(* CODESYS project jt808.20211124.1.project

Project tree, tasks and I/O mapping:
  MIC7001 : Changsha-Cyber-MI-linux, Changsha Cyber-MI Co., Ltd., version 3.5.10.40
    application Application
      libraries: Standard, * (System); CAA Types Extern, * (CAA Technical Workgroup); CAA Callback Extern, * (CAA Technical Workgroup); SysMem, * (System); SysTypes Interfaces, * (System); SysTime, * (System); CAA DTUtil Extern, 3.5.12.0 (CAA Technical Workgroup); CAA Real Time Clock Extern, 3.5.10.0 (CAA Technical Workgroup); CAN API, 1.0.0.3 (3S - Smart Software Solutions GmbH); SysFile, 3.5.15.0 (System); AC_DataLog, 3.5.14.0 (3S - Smart Software Solutions GmbH); CAA Net Base Services, 3.5.15.0 (CAA Technical Workgroup); CAA Memory, 3.5.12.0 (CAA Technical Workgroup); CAA SerialCom, 3.5.15.0 (CAA Technical Workgroup); MIC7001 base library, 1.0 (Cyber-MI.com); Util, 3.5.15.0 (System); CAA Can Low Level Imp Extern, 3.5.11.0 (CAA Technical Workgroup); CAA Can Low Level Extern, 3.5.15.0 (CAA Technical Workgroup); VisuDialogs, * (System); CmpBitmapPool, * (System); CAA File, 3.5.15.0 (CAA Technical Workgroup); IODrvEtherCAT, 3.5.15.50 (3S - Smart Software Solutions GmbH); SysShm, 3.5.8.0 (System)
      task VISU_TASK (cyclic, interval 100 ms, priority 31) calls prg_gps, prg_jt808, VisuElems.Visu_Prg
      trace Trace (task task_10ms): GVL_IO.remote_di, GVL_IO.b_mode_remote
      06_jt808/
        programs/
          program prg_jt808 [ST]: send_to_server, read_from_server, init
          program prg_gps [ST]
        Structs/
          data type stShmJT808Down
          data type stLocationExt
          data type stShmJT808Up
          data type stLocationBase
          data type stCanFrm
          data type nmeaTIME
          data type nmeaGPRMC
        functions/
          function get_sub_string_1 [ST]
          function nmea_parse_time [ST]
          function nmea_parse_date [ST]
          function get_latlon_from_str [ST]
          function nmea_parse_GPRMC [ST]
        functionblocks/
          function block Com_gps [ST]
    SoftMotion General Axis Pool
  libraries: CmpBitmapPool, * (System)
  image pool ImagePool_1
  image pool ImagePool
  5ce3da45-db07-42e7-a21c-a00fff4ed8f6|C:\Users\RJST\Desktop\bmp1.png
  text list GlobalTextList
*)

// MIC7001/Application/06_jt808/Structs/stShmJT808Down
TYPE stShmJT808Down :  // JT808下行数据
STRUCT
	location_interval:DINT;  // 位置信息发送间隔， 单位： ms
	ctrl : DINT;   // 车辆控制命令
END_STRUCT
END_TYPE

// MIC7001/Application/06_jt808/Structs/stLocationExt
TYPE stLocationExt :
STRUCT
	km_all: DINT;  // km all
	fuel:INT;   // fuel meter
	speed: INT;  // speed can
	lac:DINT; 
	cid:DINT;
	fuel_trip:DINT; // 本行程油耗
	fuel_all:DINT; 
	fuel_r_h:DINT;  // 0.05L/h
	fuel_r_l:DINT;  //  1/512Km/L
END_STRUCT
END_TYPE

// MIC7001/Application/06_jt808/Structs/stShmJT808Up
TYPE stShmJT808Up :   // 发送到服务器的上行数据
STRUCT
    location:stLocationBase;
	loc_ext:stLocationExt;
	can_data:stCanFrm;
END_STRUCT
END_TYPE

// MIC7001/Application/06_jt808/Structs/stLocationBase
TYPE stLocationBase :
STRUCT
	warning : UDINT;
    status : UDINT;
    latitude : DINT;
    longitude : DINT;
    altitude : INT;
    speed : INT;
    bearing : INT;
    asc_time :ARRAY[0..5] OF BYTE;  // ascii YYMMDDhhmmss (GMT+8)
END_STRUCT
END_TYPE

// MIC7001/Application/06_jt808/Structs/stCanFrm
TYPE stCanFrm :
STRUCT
	sn:UDINT;  // 每次更新内容后加一，用于通知底层发送程序
	id:UDINT;  //  CAN id
	data:ARRAY[0..7] OF BYTE;  // 8个字节 数据
END_STRUCT
END_TYPE

// MIC7001/Application/06_jt808/Structs/nmeaTIME
TYPE nmeaTIME :
STRUCT
	year:DINT;
	month:DINT;
	day:DINT;
	hour:DINT;
	minute:DINT;
	second:DINT;
	hsecond:DINT;
END_STRUCT
END_TYPE

// MIC7001/Application/06_jt808/Structs/nmeaGPRMC
TYPE nmeaGPRMC :
STRUCT
	utc : nmeaTIME;
	status : STRING(1);
	lat : REAL;
	ns : STRING(1);
	lon : REAL;
	ew : STRING(1);
	speed : REAL;
	direction : REAL;
	declination : REAL;
	declin_ew : STRING(1);
	mode : STRING(1);
END_STRUCT
END_TYPE

// MIC7001/Application/06_jt808/programs/prg_gps
PROGRAM prg_gps
VAR  
	filename:STRING(256) := '/tmp/connect_server.txt';
	hFile: RTS_IEC_HANDLE := 0;
	udiOpenError: RTS_IEC_RESULT;
	connect_open_flag :BOOL := TRUE;
	
	gps :Com_gps;
	com_handle :CAA.HANDLE; 
	packGPRMC : nmeaGPRMC;
	buf:STRING(255);
	gps_ok:BOOL := FALSE;
END_VAR

// 判断后端PPP网络是否连通，如果已经连通，则会同步网络时间
IF connect_open_flag THEN
	hFile := sysfileopen(szFile := filename, am := sysfile.AM_READ, pResult:= ADR(udiOpenError));
	IF hFile = RTS_INVALID_HANDLE THEN
		RETURN;
	END_IF
	
	hFile := MIC7001_BASE.close_file(hFile := hFile);
	connect_open_flag := FALSE;
END_IF

gps(xEnable := TRUE, com_hand := com_handle, gps_str => buf); 

nmea_parse_GPRMC(buf, SIZEOF(buf), ADR(packGPRMC));

IF packGPRMC.status = 'A' THEN
	gps_ok := TRUE;
ELSE
	gps_ok := FALSE;
END_IF

END_PROGRAM

// MIC7001/Application/06_jt808/functions/nmea_parse_GPRMC
FUNCTION nmea_parse_GPRMC : bool
VAR_INPUT
    buff : STRING(255);
	buff_sz : DINT;
	pack : POINTER TO nmeaGPRMC;
END_VAR
VAR
	str:STRING(255);
	rc :BOOL;
	checksum : DINT;	
END_VAR

nmea_parse_GPRMC := FALSE;

str := get_sub_string(buff, '$$', ',', 1);   //check 'GPRMC'
IF str <> 'GPRMC' THEN
	RETURN;
END_IF

//find time
str := get_sub_string(buff, ',', ',', 1);  
IF len(str) < len('hhmmss')  THEN
	RETURN;  //format error	
END_IF
IF NOT nmea_parse_time(str, ADR(pack^.utc)) THEN
	RETURN;
END_IF

//find status
str := get_sub_string(buff, ',', ',', 2);  
IF len(str)<1 THEN
	RETURN; //format error
END_IF
pack^.status := str;

//find lat
str := get_sub_string(buff, ',', ',', 3);  
IF len(str)<1 THEN
	RETURN; //format error
END_IF
pack^.lat := get_latlon_from_str(str);

//find ns
str := get_sub_string(buff, ',', ',', 4); 
IF len(str)<1 THEN
	RETURN; //format error
END_IF
pack^.ns := str;

//find lon
str := get_sub_string(buff, ',', ',', 5); 
IF len(str)<1 THEN
	RETURN; //format error
END_IF
pack^.lon := get_latlon_from_str(str);

//find ew
str := get_sub_string(buff, ',', ',', 6); 
IF len(str)<1 THEN
	RETURN; //format error
END_IF
pack^.ew := str;

//find speed
str := get_sub_string(buff, ',', ',', 7); 
IF len(str)<1 THEN
	RETURN; //format error
END_IF
pack^.speed := STRING_TO_REAL(str)*1.852;  // 节 -> km/h

//find direction
str := get_sub_string(buff, ',', ',', 8); 
IF len(str)<1 THEN
	RETURN; //format error
END_IF
pack^.direction := STRING_TO_REAL(str);

//find date
str := get_sub_string(buff, ',', ',', 9); 
IF len(str)<1 THEN
	RETURN; //format error
END_IF
IF NOT nmea_parse_date(str, ADR(pack^.utc)) THEN
	RETURN;
END_IF

//find declination
str := get_sub_string(buff, ',', ',', 10); 
IF len(str)<1 THEN
	pack^.declination := 0.0;
ELSE
	pack^.declination := STRING_TO_REAL(str);
END_IF

//find declin_ew
str := get_sub_string(buff, ',', ',', 11); 
IF len(str)<1 THEN
	RETURN; //format error
END_IF
pack^.declin_ew := str;

//find mode
str := get_sub_string(buff, ',', '*', 12); 
IF len(str) < 1 THEN
//	RETURN; // no mode is allowed
ELSE
	pack^.mode := str;
END_IF

//find checksum
str := get_sub_string(buff, '*', '$r', 1); 
IF len(str)<1 THEN
	RETURN; //format error
END_IF
checksum := STRING_TO_DINT(str);

nmea_parse_GPRMC := TRUE;

END_FUNCTION

// MIC7001/Application/06_jt808/functions/nmea_parse_time
FUNCTION nmea_parse_time : BOOL
VAR_INPUT
	str_time:STRING(255);
	p_utc:POINTER TO nmeaTIME;
END_VAR
VAR
	len_str:DINT;
END_VAR

nmea_parse_time := FALSE;

len_str := len(str_time);
IF len_str < len('hhmmss') THEN
	RETURN;  //format error
END_IF

p_utc^.hour := ANY_TO_DINT(left(str_time,2));
p_utc^.minute := ANY_TO_DINT(mid(str_time,2,3));
p_utc^.second := ANY_TO_DINT(mid(str_time,2,5));
IF len_str = len('hhmmss.u') THEN
	p_utc^.hsecond := ANY_TO_DINT(mid(str_time,1,8));
ELSIF len_str = len('hhmmss.uu') THEN
	p_utc^.hsecond := ANY_TO_DINT(mid(str_time,2,8));
ELSIF len_str = len('hhmmss.uuu') THEN
	p_utc^.hsecond := ANY_TO_DINT(mid(str_time,3,8));
ELSE
	//  no hsecond
END_IF

nmea_parse_time := TRUE;

END_FUNCTION

// MIC7001/Application/06_jt808/functions/get_latlon_from_str
FUNCTION get_latlon_from_str : REAL
VAR_INPUT
	str:STRING;
END_VAR

VAR
	temp:REAL;
	d:INT;
	m:REAL;
END_VAR

// lat format:   ddmm.mmmmmm  度度分分.分分分分分分
// lon format:  dddmm.mmmmmm  度度度分分.分分分分分分
   
temp := STRING_TO_REAL(str);
d := ANY_TO_INT(temp/100);
m := temp/100 - d;
m := m/0.6;

get_latlon_from_str := INT_TO_REAL(d)+m;

// 转换为：   度度度.度度度度度度

END_FUNCTION

// MIC7001/Application/06_jt808/functions/nmea_parse_date
FUNCTION nmea_parse_date : BOOL
VAR_INPUT
	str_time:STRING(255);
	p_utc:POINTER TO nmeaTIME;
END_VAR
VAR
	len_str:DINT;
END_VAR

nmea_parse_date := FALSE;

len_str := len(str_time);
IF len_str < len('ddmmyy') THEN
	RETURN;  //format error
END_IF

p_utc^.day := ANY_TO_DINT(left(str_time,2));
p_utc^.month := ANY_TO_DINT(mid(str_time,2,3));
p_utc^.year := ANY_TO_DINT(mid(str_time,2,5));

nmea_parse_date := TRUE;

END_FUNCTION

// MIC7001/Application/06_jt808/functionblocks/Com_gps
FUNCTION_BLOCK Com_gps
VAR_INPUT
	xEnable : BOOL := FALSE;
END_VAR
VAR_IN_OUT
	com_hand: CAA.HANDLE;
END_VAR
VAR_OUTPUT
	xDone : BOOL := FALSE;
	xError :BOOL := FALSE;
	xBusy : BOOL := FALSE;
	gps_str:STRING(255);
END_VAR
VAR
	ton_fb :TON;
	Com1Params: 			ARRAY [1..7] OF COM.PARAMETER;	(* Settings to communicate with 
the COM Port *)
	ComOpen: 				COM.Open;
	ComClose: 				COM.Close;
	ComWrite: 				COM.Write;
	ComRead: 				COM.Read;	
	Rcv_Cnt: 				CAA.SIZE;
	xCom1CloseError: 		BOOL;
	xCom1WriteError: 		BOOL;
	xCom1ReadError: 		BOOL;
	uiComState: INT := 0;
	ComID:USINT:=5;   //ttymxc4
	position :INT := 0;
	at_cmd :STRING := 'AT$r';
	at_buffer :STRING;
	ate0_cmd :STRING := 'ATE0$r';
	ate0_buffer :STRING;
	csq_cmd :STRING := 'AT+CSQ$r';
	csq_buffer :STRING;
	
	accid_cmd :STRING := 'AT+ICCID$r';
	iccid_read_buffer :STRING(255);
	ICCID_HEAD:STRING := '+ICCID: ';
	iccid:STRING(32);
	
	lac:STRING(4) := '0000';
	ci :STRING(4) := '0000';
	lac_set_cmd :STRING := 'AT+CREG=2$r';
	lac_read_cmd :STRING(255);
	
	
	lac_get_cmd :STRING := 'AT+CREG?$r';
	lac_read_buffer :STRING(255);
	
	lac_close_cmd :STRING := 'AT+CREG=0$r';
	lac_close_buffer :STRING(255);
	
	LACID_HEAD:STRING := '+CREG:';
	lac_str:STRING(8);
	ci_str:STRING(8);
	
	at_GPSCLOSE_buffer :STRING(255);
	at_GPSCLOSE_cmd :STRING := 'AT+QGPS=0$r';    
	at_GPSOPEN_cmd :STRING := 'AT+QGPS=1$r';     
	at_GPSOPEN_buffer :STRING(255);
	
	at_GPSSET_cmd :STRING := 'AT+QGPSCFG="nmeasrc",1$r';     
	at_GPSSET_buffer :STRING(255);
	
	at_GPSREAD_cmd :STRING := 'AT+QGPSGNMEA="RMC"$r';    
	at_GPSREAD_buffer :STRING(255);
	
	at_ask_buffer3 :STRING(1000);
	bit_start:INT;
	bit_end:INT;
	bit_start1:INT;
	bit_end1:INT;
	jd_info:STRING;
	wd_info:STRING;
	jd:REAL;
	wd:REAL;
	R_TIME:TIME;
	
	xDone_internal : BOOL := FALSE;
	xError_internal :BOOL := FALSE;
	
	sudu_info :STRING;
	bit_end2:INT;
	sd:REAL;
	
	ton_err:ton;
	cntr_40:DINT := 0;
END_VAR

IF NOT xEnable THEN
	xDone := FALSE;
	xError := FALSE;
	xBusy := FALSE;
	uiComState := 0;
	RETURN;
END_IF

CASE uiComState OF
	0:
	Com1Params[1].udiParameterId := COM.CAA_Parameter_Constants.udiPort;
	Com1Params[1].udiValue := ComID; 
	Com1Params[2].udiParameterId := COM.CAA_Parameter_Constants.udiBaudrate;
	Com1Params[2].udiValue := 115200;
	Com1Params[3].udiParameterId := COM.CAA_Parameter_Constants.udiParity;
	Com1Params[3].udiValue := INT_TO_UINT(COM.PARITY.NONE);
	Com1Params[4].udiParameterId := COM.CAA_Parameter_Constants.udiStopBits;
	Com1Params[4].udiValue := INT_TO_UINT(COM.STOPBIT.ONESTOPBIT);
	Com1Params[5].udiParameterId := COM.CAA_Parameter_Constants.udiTimeout;
	Com1Params[5].udiValue := 0;
	Com1Params[6].udiParameterId := COM.CAA_Parameter_Constants.udiByteSize;
	Com1Params[6].udiValue := 8;
	Com1Params[7].udiParameterId := COM.CAA_Parameter_Constants.udiBinary;
	Com1Params[7].udiValue := 0;					
	ComOpen(xExecute := TRUE, usiListLength:=UINT_TO_USINT(SIZEOF(Com1Params)/SIZEOF(COM.PARAMETER)),pParameterList:= ADR(Com1Params),hCom=> com_hand);			
	IF ComOpen.xError THEN
		ton_err(in := FALSE, pt := T#5S);
		uiComState := 32767;
	ELSIF ComOpen.xDone THEN
		uiComState := 1;
		com_hand := ComOpen.hCom;
		ComWrite(xExecute := FALSE,hCom:= com_hand);	
		ComRead(xExecute := FALSE,hCom:= com_hand);
	END_IF
	
	1:  // write "AT\r"
	ComWrite(xExecute := TRUE,hCom:= com_hand,pBuffer:= ADR(at_cmd),szSize:=len(at_cmd));		
	IF ComWrite.xError THEN
		uiComState := 200;
	END_IF
	IF ComWrite.xDone THEN
		ComWrite(xExecute := FALSE, hCom:= com_hand);
		uiComState := 2;
	END_IF
	
	2:
	ton_fb(IN := TRUE, PT := TIME#300MS);
	IF (ton_fb.Q) THEN
		ton_fb(IN := FALSE, PT := TIME#300MS);
		uiComState := 3;
	END_IF
	
	3:
	ComRead(xExecute := TRUE,hCom:= com_hand, pBuffer:= ADR(at_buffer), szBuffer:= SIZEOF(at_buffer));			
	IF ComRead.xError THEN
		uiComState := 32767;
	END_IF
	IF ComRead.xDone THEN
		position := find(at_buffer, 'OK');
		IF position > 0 THEN
			uiComState := 10;
		ELSE
			uiComState := 200;
		END_IF
		ComRead(xExecute := FALSE, hCom:= com_hand);
	END_IF
	
(*	
	4: // write "ATE0\r"
	ComWrite(xExecute := TRUE,hCom:= com_hand,pBuffer:= ADR(ate0_cmd),szSize:=len(ate0_cmd));		
	IF ComWrite.xError THEN
		uiComState := 200;
	END_IF
	IF ComWrite.xDone THEN
		ComWrite(xExecute := FALSE, hCom:= com_hand);
		uiComState := 5;
	END_IF
	
	5:
	ton_fb(IN := TRUE, PT := TIME#300MS);
	IF (ton_fb.Q) THEN
		ton_fb(IN := FALSE, PT := TIME#300MS);
		uiComState := 6;
	END_IF
	
	6:
	ComRead(xExecute := TRUE,hCom:= com_hand, pBuffer:= ADR(ate0_buffer), szBuffer:= SIZEOF(ate0_buffer));			
	IF ComRead.xError THEN
		uiComState := 200;
	END_IF
	IF ComRead.xDone THEN
		position := find(ate0_buffer, 'OK');
		IF position > 0 THEN
			uiComState := 10;
		ELSE
			uiComState := 200;
		END_IF
		ComRead(xExecute := FALSE, hCom:= com_hand);
	END_IF
	*)
	
	
	10: // write "AT+CSQ\r"
	ComWrite(xExecute := TRUE,hCom:= com_hand,pBuffer:= ADR(csq_cmd),szSize:=len(csq_cmd));		
	IF ComWrite.xError THEN
		uiComState := 200;
	END_IF
	IF ComWrite.xDone THEN
		ComWrite(xExecute := FALSE, hCom:= com_hand);
		uiComState := 11;
	END_IF
	
	11:
	ton_fb(IN := TRUE, PT := TIME#300MS);
	IF (ton_fb.Q) THEN
		ton_fb(IN := FALSE, PT := TIME#300MS);
		uiComState := 12;
	END_IF
	
	12:
	ComRead(xExecute := TRUE,hCom:= com_hand, pBuffer:= ADR(csq_buffer), szBuffer:= SIZEOF(csq_buffer));			
	IF ComRead.xError THEN
		uiComState := 200;
	END_IF
	IF ComRead.xDone THEN
		position := find(csq_buffer, 'OK');
		IF position > 0 THEN
			uiComState := 13;
		ELSE
			uiComState := 200;
		END_IF
		ComRead(xExecute := FALSE, hCom:= com_hand);
	END_IF
	
	13:
	ComWrite(xExecute := TRUE,hCom:= com_hand,pBuffer:= ADR(accid_cmd),szSize:=len(accid_cmd));		
	IF ComWrite.xError THEN
		uiComState := 200;
	END_IF
	IF ComWrite.xDone THEN
		ComWrite(xExecute := FALSE, hCom:= com_hand);
		uiComState := 14;
	END_IF
	
	14:
	ton_fb(IN := TRUE, PT := TIME#300MS);
	IF (ton_fb.Q) THEN
		ton_fb(IN := FALSE, PT := TIME#300MS);
		uiComState := 15;
	END_IF
	
	15:
	ComRead(xExecute := TRUE,hCom:= com_hand, pBuffer:= ADR(iccid_read_buffer), szBuffer:= SIZEOF(iccid_read_buffer));			
	IF ComRead.xError THEN
		uiComState := 200;
	END_IF
	IF ComRead.xDone THEN
		IF ComRead.szsize > 0 THEN
			position := find(iccid_read_buffer, ICCID_HEAD);
			IF position > 0 THEN
				iccid := mid(iccid_read_buffer, 20, position + len(ICCID_HEAD));
				uiComState := 16;
			ELSE
				uiComState := 200;
			END_IF
		ELSE
			uiComState := 200;
		END_IF
		ComRead(xExecute := FALSE, hCom:= com_hand);
	END_IF
	
	16:
	ComWrite(xExecute := TRUE,hCom:= com_hand,pBuffer:= ADR(at_GPSCLOSE_cmd),szSize:=len(at_GPSCLOSE_cmd));		
	IF ComWrite.xError THEN
		uiComState := 200;
	END_IF
	IF ComWrite.xDone THEN
		ComWrite(xExecute := FALSE, hCom:= com_hand);
		uiComState := 17;
	END_IF
	
	17:
	ton_fb(IN := TRUE, PT := TIME#300MS);
	IF (ton_fb.Q) THEN
		ton_fb(IN := FALSE, PT := TIME#300MS);
		uiComState := 18;
	END_IF
	
	18:
	ComRead(xExecute := TRUE,hCom:= com_hand, pBuffer:= ADR(at_GPSCLOSE_buffer), szBuffer:= SIZEOF(at_GPSCLOSE_buffer));			
	IF ComRead.xError THEN
		uiComState := 200;
	END_IF
	IF ComRead.xDone THEN
		uiComState := 25;
		ComRead(xExecute := FALSE, hCom:= com_hand);
	END_IF
	
	25:
	ComWrite(xExecute := TRUE,hCom:= com_hand,pBuffer:= ADR(at_GPSOPEN_cmd),szSize:= len(at_GPSOPEN_cmd));		
	IF ComWrite.xError THEN
		uiComState := 200;
	END_IF
	IF ComWrite.xDone THEN		
		ComWrite(xExecute := FALSE);
		uiComState := 26;
	END_IF
	
	26:
	ton_fb(IN := TRUE, PT := TIME#300MS);
	IF (ton_fb.Q) THEN
		ton_fb(IN := FALSE, PT := TIME#300MS);
		uiComState := 27;
	END_IF

	27:
	ComRead(xExecute := TRUE,hCom:= com_hand, pBuffer:= ADR(at_GPSOPEN_buffer), szBuffer:= SIZEOF(at_GPSOPEN_buffer));			
	IF ComRead.xError THEN
		uiComState := 200;
	END_IF
	IF ComRead.xDone THEN
		position := find(at_GPSOPEN_buffer, 'OK');
		IF position > 0 THEN
			uiComState := 28;
		ELSE
			uiComState := 200;
		END_IF
		ComRead(xExecute := FALSE, hCom:= com_hand);
	END_IF
	
	
	28:
	ComWrite(xExecute := TRUE,hCom:= com_hand,pBuffer:= ADR(at_GPSSET_cmd),szSize:= len(at_GPSSET_cmd));		//发送AT指令，查询获取的经纬度
	IF ComWrite.xError THEN
		uiComState := 200;
	END_IF
	IF ComWrite.xDone THEN		
		ComWrite(xExecute := FALSE);
		uiComState := 29;
	END_IF
	
	29:
	ton_fb(IN := TRUE, PT := TIME#300MS);
	IF (ton_fb.Q) THEN
		ton_fb(IN := FALSE, PT := TIME#300MS);
		uiComState := 30;
	END_IF
	
	30:
	ComRead(xExecute := TRUE,hCom:= com_hand, pBuffer:= ADR(at_GPSSET_buffer), szBuffer:= SIZEOF(at_GPSSET_buffer));			
	IF ComRead.xError THEN
		uiComState := 200;
	END_IF
	IF ComRead.xDone THEN
		position := find(at_GPSSET_buffer, 'OK');
		IF position > 0 THEN
			uiComState := 31;
		ELSE
			uiComState := 200;
		END_IF
		ComRead(xExecute := FALSE, hCom:= com_hand);
	END_IF
	
	
	31:
	ComWrite(xExecute := TRUE,hCom:= com_hand,pBuffer:= ADR(at_GPSREAD_cmd),szSize:= len(at_GPSREAD_cmd));		//发送AT指令，查询获取的经纬度
	IF ComWrite.xError THEN
		uiComState := 200;
	END_IF
	IF ComWrite.xDone THEN		
		ComWrite(xExecute := FALSE);
		uiComState := 32;
	END_IF

	32:
	ton_fb(IN := TRUE, PT := TIME#300MS);
	IF (ton_fb.Q) THEN
		ton_fb(IN := FALSE, PT := TIME#300MS);
		uiComState := 33;
	END_IF
	
	33:
	ComRead(xExecute := TRUE,hCom:= com_hand, pBuffer:= ADR(at_GPSREAD_buffer), szBuffer:= SIZEOF(at_GPSREAD_buffer));
	IF ComRead.xError THEN
		uiComState := 200;
	END_IF
    IF ComRead.xDone THEN
		gps_str := at_GPSREAD_buffer;
		uiComState := 40;
		cntr_40 := 0;
		ComRead(xExecute := FALSE, hCom:= com_hand);
	END_IF
	
	40:  // waiting
	   cntr_40 := cntr_40+1;
	   IF cntr_40 > 20 THEN // 2s
		   uiComState := 31;
	   END_IF
	
	200:
		xError_internal := TRUE;
		uiComState := 202;
		
	201:
		xDone_internal := TRUE;
		uiComState := 202;
		
	202:
		ComClose(xExecute := FALSE, hCom:= com_hand); 	
		uiComState := 203;
	
	203:
		ComClose(xExecute := TRUE,hCom:= com_hand);
		IF ComClose.xError THEN
			uiComState := 32767;
		END_IF
		
		IF ComClose.xDone THEN
			ComClose(xExecute := FALSE, hCom:= com_hand); 	
		
			IF xDone_internal THEN
				uiComState := 255;
			END_IF
			
			IF xError_internal THEN
				uiComState := 32767;
			END_IF
		END_IF
	
	
	255:
		xDone := TRUE;
		
	32767:	
		xError := TRUE;
		ton_err(in := TRUE, pt := T#5S);
		IF ton_err.Q THEN
			ComOpen(xExecute := FALSE, usiListLength:=UINT_TO_USINT(SIZEOF(Com1Params)/SIZEOF(COM.PARAMETER)),pParameterList:= ADR(Com1Params),hCom=> com_hand);	
			ton_err(in := FALSE, pt := T#5S);
			uiComState := 0;
		END_IF
END_CASE

END_FUNCTION_BLOCK

// MIC7001/Application/06_jt808/programs/prg_jt808
PROGRAM prg_jt808
VAR
	inited : BOOL := FALSE;
	fluidLow:INT := 0;
	lossWater:INT := 0;
	dirtyWater:INT := 0;
	littleWater:INT := 0;
	pressSuper:INT := 0;
	
	strShmFileDown : STRING := 'SHM_JT808_DW_7001';
	strShmFileUp : STRING := 'SHM_JT808_UP_7001';
	hShMemDown: RTS_IEC_HANDLE := RTS_INVALID_HANDLE ;
	hShMemUp: RTS_IEC_HANDLE := RTS_INVALID_HANDLE ;
	ResultRead: RTS_IEC_RESULT;
	ResultWrite: RTS_IEC_RESULT;
	
	iRead: __UXINT;
	iWrite: __UXINT;
	shmDataDown:stShmJT808Down;
	shmDataUp:stShmJT808Up;
	sizeOfStFromAliyun:__UXINT := SIZEOF(stShmJT808Down);
	sizeOfStToAliyun:__UXINT := SIZEOF(stShmJT808Up);
	
	sim_data : DINT := 0;
	digi_val :DWORD := 0;
	lock_1 :BOOL := FALSE;
	lock_2 :BOOL := FALSE;
	unlock :BOOL := FALSE;
	test_val2 :DINT;
	
	get_dt:dtu.GetDateandTime();
	tempdt : DWORD;
	g_uiYear:UINT;
	g_uiMonth:UINT;
	g_uiDate:UINT;
	g_uiHour:UINT;
	g_uiMinute:UINT;
	g_uiSecond:UINT;
END_VAR


IF NOT inited THEN
 	IF NOT init() THEN  // 初始化失败
		RETURN;
	ELSE
		inited := TRUE;
		
		sim_data := 0;
		test_val2 := 0;
	END_IF  
END_IF

IF read_from_server() THEN
   // 读取阿里云发来的数据
	IF shmDataDown.ctrl > 0 THEN
		// 处理命令通道1
	END_IF
END_IF

// 准备上传到阿里云的数据
sim_data := sim_data + 1;

get_dt(xExecute := TRUE);
 IF get_dt.xDone THEN
  tempdt := DT_TO_DWORD(get_dt.dtDateandtime);
  tempdt := tempdt + 3600*8;   // utc 时间转为北京时间
  dtu.DTSplit(DWORD_TO_DT(tempdt), ADR(g_uiYear), ADR(g_uiMonth), ADR(g_uiDate), ADR(g_uiHour), ADR(g_uiMinute), ADR(g_uiSecond));

  get_dt(xExecute := FALSE);

 END_IF

shmDataUp.location.asc_time[0] := ANY_TO_BYTE(g_uiYear MOD 100);
shmDataUp.location.asc_time[1] := ANY_TO_BYTE(g_uiMonth);
shmDataUp.location.asc_time[2] := ANY_TO_BYTE(g_uiDate);
shmDataUp.location.asc_time[3] := ANY_TO_BYTE(g_uiHour);
shmDataUp.location.asc_time[4] := ANY_TO_BYTE(g_uiMinute);
shmDataUp.location.asc_time[5] := ANY_TO_BYTE(g_uiSecond);

shmDataUp.loc_ext.km_all := ANY_TO_DINT( gvl_es.trip_all_1939*10);      // jt808 unit: 0.1Km
shmDataUp.loc_ext.fuel_trip := ANY_TO_DINT(gvl_es.fuel_trip_engine*2);  // jt808 unit: 0.5L
shmDataUp.loc_ext.fuel_all := ANY_TO_DINT( gvl_es.fuelall_engine*2);    // jt808 unit: 0.5L
shmDataUp.loc_ext.fuel_r_h := ANY_TO_DINT(gvl_es.fuelrate_engine*20);   // jt808 unit: 0.05L/h
IF gvl_es.fuel_100km = 0 OR gvl_es.fuel_100km = 999 THEN
	shmDataUp.loc_ext.fuel_r_l := 0;
ELSE
	shmDataUp.loc_ext.fuel_r_l := ANY_TO_DINT(512*100/gvl_es.fuel_100km);   // jt808 unit: 1/512Km/L
END_IF

IF prg_gps.packGPRMC.status = 'A' THEN  // GPS定位成功
	shmDataUp.location.latitude := ANY_TO_DINT(prg_gps.packGPRMC.lat*1000000);
	shmDataUp.location.longitude := ANY_TO_DINT(prg_gps.packGPRMC.lon*1000000);
	shmDataUp.location.altitude := 54;
	shmDataUp.location.speed := ANY_TO_INT(prg_gps.packGPRMC.speed);
	shmDataUp.location.bearing := ANY_TO_INT(prg_gps.packGPRMC.direction);
	shmDataUp.location.status := 16#03;   
ELSIF 	prg_gps.packGPRMC.status = 'V' THEN  // 有GPS，但尚未定位成功
	shmDataUp.location.latitude := 0;
	shmDataUp.location.longitude := 0;	
	shmDataUp.location.altitude := 0;
	shmDataUp.location.speed := 0;
	shmDataUp.location.bearing := 0;	
	shmDataUp.location.status := 16#02;   
ELSE	// 没有GPS
    shmDataUp.loc_ext.lac := MIC7001_base.read_num_from_file(filename := '/tmp/lac.txt');
	shmDataUp.loc_ext.cid := MIC7001_base.read_num_from_file(filename := '/tmp/cid.txt');
	shmDataUp.location.latitude := 28230306;
	shmDataUp.location.longitude := 113414176;	
	shmDataUp.location.altitude := 0;	
	shmDataUp.location.status := 16#03;   
END_IF

IF send_to_server() THEN
	// write ok
END_IF

METHOD send_to_server : bool
VAR_INPUT
END_VAR
send_to_server := FALSE;

iWrite := sysshm.SysSharedMemoryWrite(hShMemUp, 0, ADR(shmDataUp), sizeOfStToAliyun, ADR(ResultWrite));
IF iWrite = sizeOfStToAliyun THEN
	send_to_server := TRUE;
END_IF

RETURN;
END_METHOD

METHOD read_from_server : bool
VAR_INPUT
END_VAR
read_from_server := FALSE;

iRead := sysshm.SysSharedMemoryRead(hShMemDown, 0, ADR(shmDataDown), sizeOfStFromAliyun, ADR(ResultRead));
IF iRead = sizeOfStFromAliyun THEN
    read_from_server := TRUE;
END_IF

RETURN;
END_METHOD

METHOD init : bool
VAR_INPUT
END_VAR
init := FALSE;

IF hShMemDown = RTS_INVALID_HANDLE  THEN
	hShMemDown := sysshm.SysSharedMemoryCreate(strShmFileDown, 0, ADR(sizeOfStFromAliyun), ADR(ResultRead));	
END_IF

IF hShMemUp = RTS_INVALID_HANDLE  THEN
	hShMemUp := sysshm.SysSharedMemoryCreate(strShmFileUp, 0, ADR(sizeOfStToAliyun), ADR(ResultRead));	
END_IF

IF hShMemDown = RTS_INVALID_HANDLE  OR hShMemUp = RTS_INVALID_HANDLE  THEN
	RETURN;
END_IF

init := TRUE;
RETURN;
END_METHOD

END_PROGRAM

// MIC7001/Application/06_jt808/functions/get_sub_string_1
FUNCTION get_sub_string_1 : string(255)
VAR_INPUT
	in_str : STRING(255);
	char_l : STRING(1);
	char_r : STRING(1);
	index : DINT := 1;
END_VAR
VAR
	start : DINT;
	end : DINT;
	sub_str : STRING(255);
	length : DINT;
	i :DINT;
END_VAR

get_sub_string := '';
sub_str := in_str;
i := index;

length := len(sub_str);
start := 0;
end := length+1;

WHILE i > 0 DO
	start := find(sub_str, char_l);
	IF start = 0 THEN
		RETURN;
	END_IF
	sub_str := right(sub_str, DINT_TO_INT(length-start));
	length := len(sub_str);
	i := i - 1;
END_WHILE

end := find(sub_str, char_r);
IF end = 0 THEN
	end := length + 1;
END_IF
get_sub_string := left(sub_str, DINT_TO_INT(end-1));

END_FUNCTION
